// TIA Portal V20 export
DATA_BLOCK "LBP_OpUnitComm_DB"   // DB70
// stored: InstanceOfName LBP_OpUnitComm, InstanceOfType FB
"LBP_OpUnitComm"
   // VAR_OUTPUT
   //    Error : Bool;
   //    Status : Word;
   // END_VAR
   // VAR_IN_OUT
   //    Config : Variant;
   // END_VAR
   // VAR
   //    s_OpUnitConnInstance { S7_SetPoint := 'True'} : Array[1..6] of "LBP_InternalProc2";
   //    s_OpUnitNumber : UInt;
   //    s_OpUnitHardwareInterfaceId : HW_ANY;
   //    s_OpUnitEnabled : Array[1..6] of Bool;
   //    s_OpUnitConfig { S7_SetPoint := 'True'} : Array[1..6] of "LBP_typeInternal1";
   //    s_OpUnitControlMcp : Array[1..5] of Struct
   //       active : Bool;
   //       stop : Bool;
   //       notSend : Bool;
   //       connected : Bool;
   //       warning : Bool;
   //       error : Bool;
   //       status : Word;
   //       info : Word;
   //       alert : Bool;
   //       alertDelay { S7_SetPoint := 'True'} : TON_TIME;
   //    END_STRUCT;
   //    s_OpUnitControlIdent : Struct
   //       strobe : Bool;
   //       busAddress : USInt;
   //       modeDck : Bool;
   //       numberOfInputBytes : UInt;
   //       numberOfOutputBytes : UInt;
   //       mcpType : Word;
   //       done : Bool;
   //       error : Bool;
   //       status : Word;
   //       info : Word;
   //    END_STRUCT;
   //    s_OpUnitData : Array[1..6] of Struct
   //       connect : Bool;
   //       ident : Bool;
   //       notSend : Bool;
   //       busy : Bool;
   //       connected : Bool;
   //       warning : Bool;
   //       error : Bool;
   //       identReady : Bool;
   //       reconnect : Bool;
   //       status : Word;
   //       errorInfo : Word;
   //       mcpType : Word;
   //       mcpDipFixes : Word;
   //       numberOfOutputBytes : UInt;
   //       numberOfInputBytes : UInt;
   //       numberOfHandwheels : UInt;
   //       handwheelRecent : Bool;
   //       handwheelPulses1 : Int;
   //       handwheelPulses2 : Int;
   //       handwheelStopped1 : Bool;
   //       handwheelStopped2 : Bool;
   //       reconnectTimer { S7_SetPoint := 'True'} : TON_TIME;
   //       reconnectCounter : UInt;
   //    END_STRUCT;
   //    s_init : Bool;
   //    statReadWriteRecordActive : Bool;
   //    statReadWriteRecordComplete : Bool;
   //    statReadWriteRecordAbort : Bool;
   //    statReadWriteRecordMcp : UInt;
   //    statReadWriteRecordTimeout : TON_TIME;
   //    statReadWriteRecordData { S7_SetPoint := 'True'} : "LBP_typeInternal5";
   // END_VAR
BEGIN
END_DATA_BLOCK
